FUNCTION_BLOCK TEvent_ExecutionAborted EXTENDS TEventBase IMPLEMENTS IEvent
VAR
    Message : T_MaxString;
    Handler : IEventHandler_OnExecutionAborted;
END_VAR

METHOD  CallHandler
VAR_INPUT
    HandlerBase : IEventHandlerBase;
    EventArgs   : IStreamReader;
END_VAR
VAR
    Message : T_MaxString;
END_VAR
IF __QUERYINTERFACE(HandlerBase,Handler) THEN
    Message := EventArgs.Read_STRING();
    Handler.OnExecutionAborted(Message);
END_IF
END_METHOD

METHOD  IsHandlerSupported : BOOL
VAR_INPUT
    HandlerBase : IEventHandlerBase;
END_VAR
IF __QUERYINTERFACE(HandlerBase,Handler) THEN
    IsHandlerSupported := TRUE;
END_IF
END_METHOD

END_FUNCTION_BLOCK

(* stored: Version 1.1.0.1, ProductVersion 3.1.4024.3
   POU TEvent_ExecutionAborted: Id {b45b5c98-1cf5-4828-b823-eb7ae1050611}, SpecialFunc None
   Method CallHandler: Id {710150a8-2630-4352-a2f2-4c852696e948}
   Method IsHandlerSupported: Id {36f5197e-0951-47ff-a35b-d6f696eb71ef} *)
